// Load stacker HW inputs
TYPE ST_InputsLoadstacker :
STRUCT	
	HW				: ST_HW_InputsLoadstacker;	// Hardware inputs
	CtrlIn			: ST_CtrlInLoadstacker;		// ser function control inputs	
END_STRUCT
END_TYPE

(* stored: Version 1.1.0.1, ProductVersion 3.1.4024.4
   DUT ST_InputsLoadstacker: Id {623ed4fa-46d0-472c-bdac-bc3299812848} *)
